// TwinCAT 3 PLC project ADS_communication
// ProgramVersion: 3.1.4024.0
// libraries:
//   Tc2_EtherCAT, * (Beckhoff Automation GmbH)
//   Tc2_MC2, * (Beckhoff Automation GmbH)
//   Tc2_NC, * (Beckhoff Automation GmbH)
//   Tc2_Standard, * (Beckhoff Automation GmbH)
//   Tc2_System, * (Beckhoff Automation GmbH)
//   Tc3_Module, * (Beckhoff Automation GmbH)
//   VisuDialogs, * (System)
// project tree:
//   / GlobalTextList.TcGTLO, PlcTask.TcTTO, Visualization Manager.TcVMO (not stored)
//   POUs/ MAIN.TcPOU
//   VISUs/ Visualization.TcVIS
// real-time tasks:
//   TASK PlcTask: cycle T#10ms, priority 20, ADS port 350
// motion (NC):
//   TASK NC-Task 1 SAF: cycle T#2ms, priority 4, ADS port 501
//   TASK NC-Task 1 SVB: cycle T#10ms, priority 8, ADS port 511
//   AXIS MotorOne (id 1)
//     OtherSettings: AllowMotionCmdToSlave=true
//     encoder EncType=19
//       EncPara: MaxCount=#xffffffff
//     drive DrvType=16
//       DrvPara: MaxCount=#xffffffff, DriveControlDWord=#x00020000
//         Analog: TorqueSetpointScale=10, ScaleFactorActTorque=0.1
//         TimeComp: TaskDelayCycles=1
//     controller CtrType=1
//       CtrPara: PriorControlFactor=1
//         Observer: BandWidth=20
//   AXIS MotorTwo (id 2)
//     OtherSettings: AllowMotionCmdToSlave=true
//     encoder EncType=19
//       EncPara: MaxCount=#xffffffff
//     drive DrvType=16
//       DrvPara: MaxCount=#xffffffff, DriveControlDWord=#x00020000
//         Analog: TorqueSetpointScale=10, ScaleFactorActTorque=0.1
//         TimeComp: TaskDelayCycles=1
//     controller CtrType=1
//       CtrPara: PriorControlFactor=1
//         Observer: BandWidth=20
// I/O:
//   DEVICE Device 3 (EtherCAT), AmsNetId 10.0.20.83.4.1
//     Drive 1 (Servo 9400 Highline TA CiA 402) [Servo 9400 Highline ECAT V3 TA CiA 402]
//     Drive 2 (Servo 9400 Highline TA CiA 402) [Servo 9400 Highline ECAT V2 TA CiA 402]
// variable links:
//   NC-Task 1 SAF/Axes/MotorOne <-> Device 3 (EtherCAT)/Drive 1 (Servo 9400 Highline TA CiA 402)
//     Drive/Inputs/In/nState1 <-> Cylic Position Mode/Statusword
//     Drive/Inputs/In/nState2 <-> Cylic Position Mode/Statusword @bit 8
//     Drive/Inputs/In/nState4 @bit 1 <-> WcState/InputToggle
//     Drive/Inputs/In/nState4 <-> WcState/WcStateIn
//     Drive/Inputs/In/nState5 <-> Cylic Position Mode/Mode of Operation display
//     Drive/Outputs/Out/nCtrl1 <-> Cylic Position Mode_1/Controlword
//     Drive/Outputs/Out/nCtrl2 <-> Cylic Position Mode_1/Controlword @bit 8
//     Drive/Outputs/Out/nCtrl5 <-> Cylic Position Mode_1/Mode of Operation
//     Drive/Outputs/Out/nDataOut1 <-> Cylic Position Mode_1/Target position
//     Enc/Inputs/In/nDataIn1 <-> Cylic Position Mode/Position actual value (units)
//     Enc/Inputs/In/nState4 @bit 1 <-> WcState/InputToggle
//     Enc/Inputs/In/nState4 <-> WcState/WcStateIn
//   NC-Task 1 SAF/Axes/MotorTwo <-> Device 3 (EtherCAT)/Drive 2 (Servo 9400 Highline TA CiA 402)
//     Drive/Inputs/In/nState1 <-> Cylic Position Mode/Statusword
//     Drive/Inputs/In/nState2 <-> Cylic Position Mode/Statusword @bit 8
//     Drive/Inputs/In/nState4 @bit 1 <-> WcState/InputToggle
//     Drive/Inputs/In/nState4 <-> WcState/WcStateIn
//     Drive/Inputs/In/nState5 <-> Cylic Position Mode/Mode of Operation display
//     Drive/Outputs/Out/nCtrl1 <-> Cylic Position Mode_1/Controlword
//     Drive/Outputs/Out/nCtrl2 <-> Cylic Position Mode_1/Controlword @bit 8
//     Drive/Outputs/Out/nCtrl5 <-> Cylic Position Mode_1/Mode of Operation
//     Drive/Outputs/Out/nDataOut1 <-> Cylic Position Mode_1/Target position
//     Enc/Inputs/In/nDataIn1 <-> Cylic Position Mode/Position actual value (units)
//     Enc/Inputs/In/nState4 @bit 1 <-> WcState/InputToggle
//     Enc/Inputs/In/nState4 <-> WcState/WcStateIn

CONFIGURATION ADS_communication
    RESOURCE PLC ON TwinCAT3
        TASK PlcTask(INTERVAL := T#10ms, PRIORITY := 20);
        PROGRAM MAIN WITH PlcTask : MAIN;
    END_RESOURCE
END_CONFIGURATION

// ---- POUs/MAIN.TcPOU
PROGRAM MAIN
VAR
	fbReadRequest : ADSREAD; //send request
	fbWriteRequest : ADSWRITE; //recive answer
	fbWriteValue : ADSWRITE; //write based on the answer
	bRequestToWrite : BOOL; //when set to true we request to write a variable
	bAnswerToRequest : BOOL; //we read the answer from the PLC where the process is ongoing
	rValueToWrite : LREAL; //we write the value to the other PLC
	
	fbTimerToRead : TON; //timer for reading the request
	fbTimerToReadSDO : TON; //timer for reading sdo 
	
	fbSdoRead : FB_EcCoeSdoRead; //sdo read function block
	ActPosSDO : DINT; //buffer where to position value will be stored
END_VAR

fbTimerToRead.IN := NOT fbTimerToRead.Q; //timer to read the request
fbTimerToReadSDO.IN := NOT fbTimerToReadSDO.Q;

fbWriteRequest(NetId := '169.254.154.248.1.1', //requesting to write a value to the PLC
		Port := 851,
		IDXGRP := 16#4040,
		IDXOFFS := 385000,
		LEN := SIZEOF(bRequestToWrite),
		SRCADDR := ADR(bRequestToWrite),
		Write := bRequestToWrite);
		
fbReadRequest(NetId := '169.254.154.248.1.1', //reading the answer to the request
	   Port := 851, 
	   IDXGRP := 16#4040,
	   IDXOFFS := 385008,
	   LEN := SIZEOF(bAnswerToRequest),
	   DESTADDR := ADR(bAnswerToRequest),
	   Read := fbTimerToRead.Q);

		
fbWriteValue(NetId := '169.254.154.248.1.1', //writing the value after the request has been approved
		Port := 851,
		IDXGRP := 16#4040,
		IDXOFFS :=447616,
		LEN := SIZEOF(rValueToWrite),
		SRCADDR := ADR(rValueToWrite),
		Write := bAnswerToRequest);

fbSdoRead(sNetId := '10.0.20.83.4.1', //reading the position of the motor as SDO
		nSlaveAddr := 1001,
		nIndex := 16#6064,
		nSubIndex := 0,
		cbBufLen := SIZEOF(ActPosSDO),
		pDstBuf := ADR(ActPosSDO),
		bExecute := fbTimerToReadSDO.Q);
		
fbTimerToRead(PT := T#2S);
fbTimerToReadSDO(PT := T#500MS);

END_PROGRAM

// ---- GlobalTextList.TcGTLO
TEXTLIST GlobalTextList
  393 = '%f'
  361 = 'Value to request: %f'
END_TEXTLIST

// ---- VISUs/Visualization.TcVIS
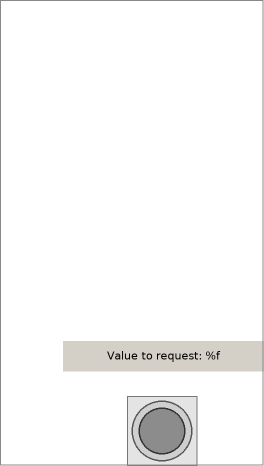
VISUALIZATION Visualization  // 264x466
    Textfield (63,341 201x30), "Value to request: %f", text variable: MAIN.rValueToWrite
        OnMouseClick: write MAIN.rValueToWrite via Default
    PushSwitch (127,396 70x70), variable: MAIN.bRequestToWrite, behaviour: TAP, style: Switch-PushSwitch-Gray
END_VISUALIZATION
